// Checks if a generic is time.
FUNCTION F_Is_Time_Generic : BOOL
VAR_INPUT
	Value : T_Generic;
END_VAR
VAR
END_VAR

CASE Value.TypeClass OF
	__SYSTEM.TYPE_CLASS.TYPE_TIME,
	__SYSTEM.TYPE_CLASS.TYPE_LTIME,
	__SYSTEM.TYPE_CLASS.TYPE_TIMEOFDAY:
		F_Is_Time_Generic := TRUE;
END_CASE

END_FUNCTION

(* stored: Version 1.1.0.1, ProductVersion 3.1.4024.4
   POU F_Is_Time_Generic: Id {ba410df6-6f3b-0467-332a-fe1604d0370d}, SpecialFunc None *)
